{attribute 'GeneratedUsingTerminal: EL7332-0000-0016'}
{attribute addProperty BoxType "EL7332-0000-0016"}
{attribute addProperty Id "ControlAT %Q*Control_C948E0F23"}
{attribute addProperty CRC "1519079446"}
{attribute addProperty Size "3"}
TYPE DCM_Control_Channel_5A8B5016 :
STRUCT
	{attribute addProperty Name "Control"}
	Control AT %Q* : Control_C948E0F2;
END_STRUCT
END_TYPE

(* stored: Version 1.2.0.0, ProductVersion 3.1.4024.9
   DUT DCM_Control_Channel_5A8B5016: Id {6809cb00-4599-438c-ae21-8882bce31224} *)
